(* Logix 5000 project; controller Lab8_2 5069-L306ERM rev 35.11; software revision 35.03 *)

TASK MainTask (continuous, watchdog 500 ms) : MainProgram

MODULES
   Local : 5069-L306ERM (5069 0, rev 35.11)
      IOHub : vendor 1 type 7 code 358 (Ethernet 192.168.105.5, rev 1.1, Output RPI 20 ms)
END_MODULES

PROGRAM MainProgram   (* main routine Lab8_2 *)
VAR
   decrypted : BOOL;
   enabled : BOOL;
   enabled_0 : BOOL;
   enabled_2 : BOOL;
   enabled_2_4 : BOOL;
   enabled_4 : BOOL;
   encrypted : BOOL;
   i : DINT;
   MrArray : DINT[64];
   MrString : STRING;
   shift : DINT;
   shifted : BOOL;
END_VAR

ROUTINE Lab8_2   (* structured text *)
   // RisingEdge:= R_TRIG
   // RisingEdge(CLK:= IOHub:I.Data.0)
   
   // JSR()
   
   
   // rising edge helper
   if not IOHub:I.Data.0 then
   	enabled_0:= 1;
   end_if;
   
   if not IOHub:I.Data.2 then
   	enabled_2:= 1;
   end_if;
   
   /*
   if not IOHub:I.Data.4 then
   	enabled_4:= 1;
   end_if;
   
   if not IOHub:I.Data.2 and not IOHub:I.Data.4 then
   	enabled_2_4:= 1;
   end_if;
   
   */
   
   // get shift value
   if IOHub:I.Data.0 then
   	if enabled_0 then
   		shift:= shift + 1;
   		enabled_0:= 0;
   	end_if;
   end_if;
   
   // load
   if IOHub:I.Data.2 then
   	if enabled_2 then
   		for i:= 0 to MrString.LEN by 1 do
   			MrArray[i]:= MrString.DATA[i];
   		end_for;
   		enabled_2:= 0;
   	end_if;
   end_if;
   
   // shift (encryption)
   if IOHub:I.Data.4 then
   	if not encrypted then
   		shifted:= 1;
   		for i:= 0 to MrString.LEN by 1 do
   			MrArray[i]:= MrArray[i] + shift;
   		end_for;
   		encrypted:= 1;
   	end_if;
   end_if;
   
   // decryption
   if IOHub:I.Data.2 and IOHub:I.Data.4 then
   	if encrypted then
   		for i:= 0 to MrString.LEN by 1 do
   			MrArray[i]:= MrArray[i] - shift;
   		end_for;
   		encrypted:= 0;
   	end_if;
   end_if;
   
   
   
   
   
   
   
END_ROUTINE
END_PROGRAM
